{attribute 'qualified_only'}
{attribute 'strict'}
TYPE E_MOTOR_RPC_ERROR :
(
	OK						:= 0,
	NOT_OP					:= -1,			
	NOT_NOTOP_READY			:= -2,			
	NOT_NOTOP_NOTREADY		:= -3,			
	LOCAL					:= -4,			
	SW_LIMIT_LOWER			:= -5,			
	SW_LIMIT_UPPER			:= -6,			
	INIT_WHILE_MOVING		:= -7,
	VEL_ZERO				:= -8,			
	VEL_NEG					:= -9,			
	VEL_MAX					:= -10,

	UNSAFE					:= -11	// EICSSW-1923			
);
END_TYPE

(* stored: Version 1.1.0.1, ProductVersion 3.1.4024.12
   DUT E_MOTOR_RPC_ERROR: Id {ae0abd72-7773-43bc-83e5-11d973ea74e5} *)
